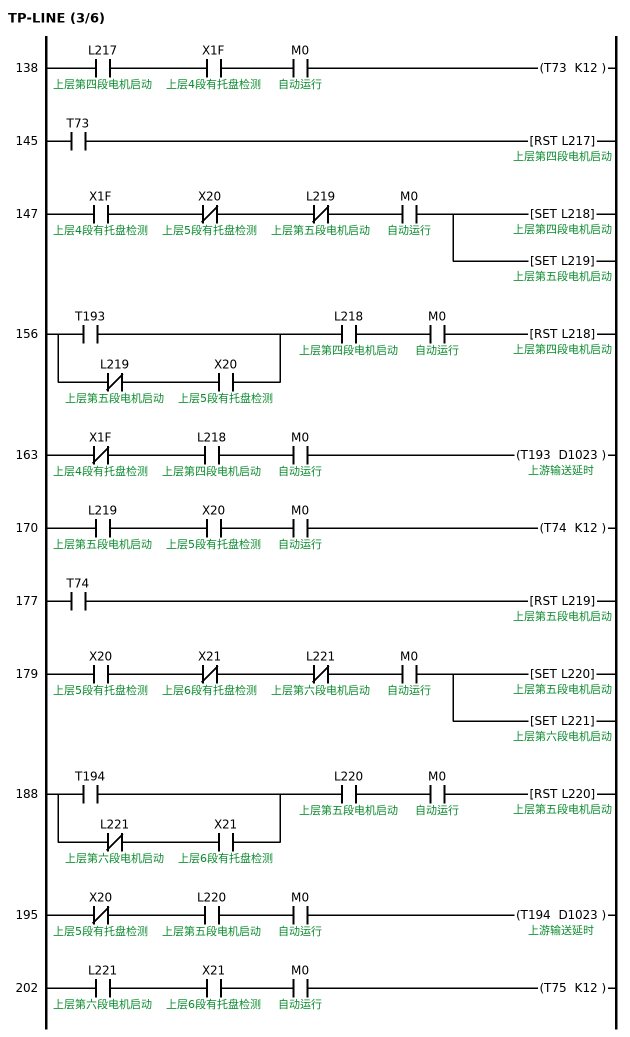
[picture p72: ladder of TP-LINE, rungs at steps 138 to 202]
138   LD      L217  ; 上层第四段电机启动
      AND     X1F  ; 上层4段有托盘检测
      AND     M0  ; 自动运行
      OUT     T73 K12
145   LD      T73
      RST     L217  ; 上层第四段电机启动
147   LD      X1F  ; 上层4段有托盘检测
      ANI     X20  ; 上层5段有托盘检测
      ANI     L219  ; 上层第五段电机启动
      AND     M0  ; 自动运行
      SET     L218  ; 上层第四段电机启动
        [note] 5
      SET     L219  ; 上层第五段电机启动
156   LD      T193
      LDI     L219  ; 上层第五段电机启动
      AND     X20  ; 上层5段有托盘检测
      ORB
      AND     L218  ; 上层第四段电机启动
      AND     M0  ; 自动运行
      RST     L218  ; 上层第四段电机启动
163   LDI     X1F  ; 上层4段有托盘检测
      AND     L218  ; 上层第四段电机启动
      AND     M0  ; 自动运行
      OUT     T193 D1023  ; 上游输送延时
170   LD      L219  ; 上层第五段电机启动
      AND     X20  ; 上层5段有托盘检测
      AND     M0  ; 自动运行
      OUT     T74 K12
177   LD      T74
      RST     L219  ; 上层第五段电机启动
179   LD      X20  ; 上层5段有托盘检测
      ANI     X21  ; 上层6段有托盘检测
      ANI     L221  ; 上层第六段电机启动
      AND     M0  ; 自动运行
      SET     L220  ; 上层第五段电机启动
        [note] 6
      SET     L221  ; 上层第六段电机启动
188   LD      T194
      LDI     L221  ; 上层第六段电机启动
      AND     X21  ; 上层6段有托盘检测
      ORB
      AND     L220  ; 上层第五段电机启动
      AND     M0  ; 自动运行
      RST     L220  ; 上层第五段电机启动
195   LDI     X20  ; 上层5段有托盘检测
      AND     L220  ; 上层第五段电机启动
      AND     M0  ; 自动运行
      OUT     T194 D1023  ; 上游输送延时
202   LD      L221  ; 上层第六段电机启动
      AND     X21  ; 上层6段有托盘检测
      AND     M0  ; 自动运行
      OUT     T75 K12
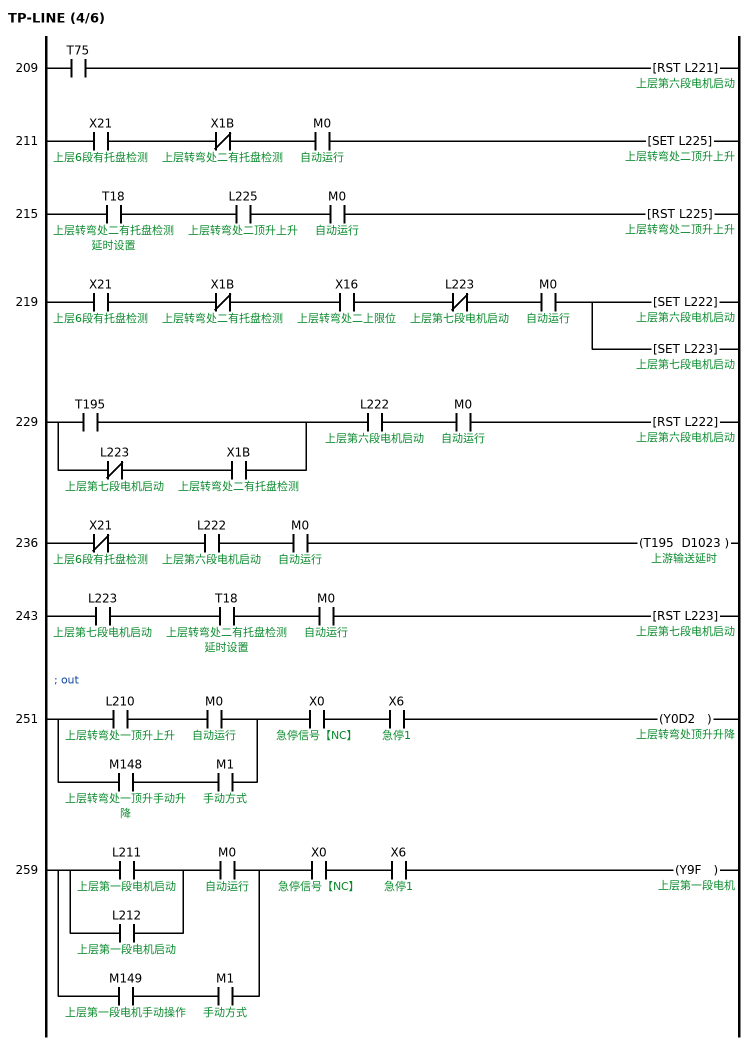
209   LD      T75
      RST     L221  ; 上层第六段电机启动
211   LD      X21  ; 上层6段有托盘检测
      ANI     X1B  ; 上层转弯处二有托盘检测
      AND     M0  ; 自动运行
      SET     L225  ; 上层转弯处二顶升上升
215   LD      T18  ; 上层转弯处二有托盘检测延时设置
      AND     L225  ; 上层转弯处二顶升上升
      AND     M0  ; 自动运行
      RST     L225  ; 上层转弯处二顶升上升
219   LD      X21  ; 上层6段有托盘检测
      ANI     X1B  ; 上层转弯处二有托盘检测
      AND     X16  ; 上层转弯处二上限位
      ANI     L223  ; 上层第七段电机启动
      AND     M0  ; 自动运行
      SET     L222  ; 上层第六段电机启动
        [note] 7
      SET     L223  ; 上层第七段电机启动
229   LD      T195
      LDI     L223  ; 上层第七段电机启动
      AND     X1B  ; 上层转弯处二有托盘检测
      ORB
      AND     L222  ; 上层第六段电机启动
      AND     M0  ; 自动运行
      RST     L222  ; 上层第六段电机启动
236   LDI     X21  ; 上层6段有托盘检测
      AND     L222  ; 上层第六段电机启动
      AND     M0  ; 自动运行
      OUT     T195 D1023  ; 上游输送延时
243   LD      L223  ; 上层第七段电机启动
      AND     T18  ; 上层转弯处二有托盘检测延时设置
      AND     M0  ; 自动运行
      RST     L223  ; 上层第七段电机启动
; out
251   LD      L210  ; 上层转弯处一顶升上升
      AND     M0  ; 自动运行
      LD      M148  ; 上层转弯处一顶升手动升降
      AND     M1  ; 手动方式
      ORB
      AND     X0  ; 急停信号【NC】
      AND     X6  ; 急停1
      OUT     Y0D2  ; 上层转弯处顶升升降
259   LD      L211  ; 上层第一段电机启动
      OR      L212  ; 上层第一段电机启动
      AND     M0  ; 自动运行
      LD      M149  ; 上层第一段电机手动操作
      AND     M1  ; 手动方式
      ORB
      AND     X0  ; 急停信号【NC】
      AND     X6  ; 急停1
      OUT     Y9F  ; 上层第一段电机
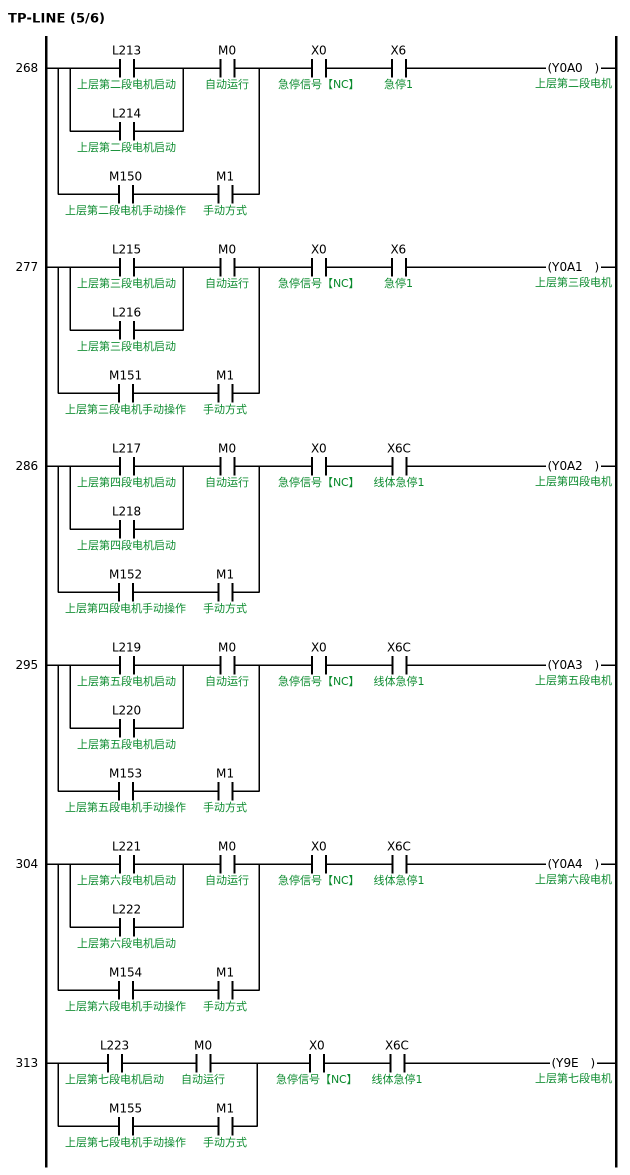
268   LD      L213  ; 上层第二段电机启动
      OR      L214  ; 上层第二段电机启动
      AND     M0  ; 自动运行
      LD      M150  ; 上层第二段电机手动操作
      AND     M1  ; 手动方式
      ORB
      AND     X0  ; 急停信号【NC】
      AND     X6  ; 急停1
      OUT     Y0A0  ; 上层第二段电机
277   LD      L215  ; 上层第三段电机启动
      OR      L216  ; 上层第三段电机启动
      AND     M0  ; 自动运行
      LD      M151  ; 上层第三段电机手动操作
      AND     M1  ; 手动方式
      ORB
      AND     X0  ; 急停信号【NC】
      AND     X6  ; 急停1
      OUT     Y0A1  ; 上层第三段电机
286   LD      L217  ; 上层第四段电机启动
      OR      L218  ; 上层第四段电机启动
      AND     M0  ; 自动运行
      LD      M152  ; 上层第四段电机手动操作
      AND     M1  ; 手动方式
      ORB
      AND     X0  ; 急停信号【NC】
      AND     X6C  ; 线体急停1
      OUT     Y0A2  ; 上层第四段电机
295   LD      L219  ; 上层第五段电机启动
      OR      L220  ; 上层第五段电机启动
      AND     M0  ; 自动运行
      LD      M153  ; 上层第五段电机手动操作
      AND     M1  ; 手动方式
      ORB
      AND     X0  ; 急停信号【NC】
      AND     X6C  ; 线体急停1
      OUT     Y0A3  ; 上层第五段电机
304   LD      L221  ; 上层第六段电机启动
      OR      L222  ; 上层第六段电机启动
      AND     M0  ; 自动运行
      LD      M154  ; 上层第六段电机手动操作
      AND     M1  ; 手动方式
      ORB
      AND     X0  ; 急停信号【NC】
      AND     X6C  ; 线体急停1
      OUT     Y0A4  ; 上层第六段电机
313   LD      L223  ; 上层第七段电机启动
      AND     M0  ; 自动运行
      LD      M155  ; 上层第七段电机手动操作
      AND     M1  ; 手动方式
      ORB
      AND     X0  ; 急停信号【NC】
      AND     X6C  ; 线体急停1
      OUT     Y9E  ; 上层第七段电机
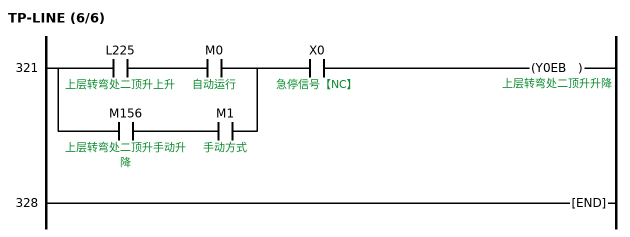
321   LD      L225  ; 上层转弯处二顶升上升
      AND     M0  ; 自动运行
      LD      M156  ; 上层转弯处二顶升手动升降
      AND     M1  ; 手动方式
      ORB
      AND     X0  ; 急停信号【NC】
      OUT     Y0EB  ; 上层转弯处二顶升升降
328   END
END_PROGRAM

PROGRAM ServoScan
VAR
  istep : INT;  (* 扫码步骤 *)
END_VAR
VAR CONSTANT
  ROW : INT := 8;  (* Y轴每个值对应的电池数量 *)
END_VAR
VAR
  ii : INT;
  jj : INT;
  m_xclean : BOOL;  (* 清零 *)
  kk : INT;  (* 错误位 *)
END_VAR

(*报警信息读取*)
g_iXanisAlarm:=U10\G806;
g_iYanisAlarm:=U10\G906;
(*报警复位*)
IF LDP(TRUE,g_xResetServo) THEN
	U10\G1502:=1;(*X轴复位*)(*这俩信号都能自动复位*)
	U10\G1602:=1;(*Y轴复位*)
	U10\G1503:=1;(*X轴重起*)
	U10\G1603:=1;(*Y轴重起*)
	YBE:= X78 OR  X79;(*X78,X79为两个驱动器的报警，这个驱动器只能断电复位，所以YAE控制断电*)
ELSIF LDF(TRUE,g_xResetServo)THEN
	YBE:=0;
END_IF;	







(*下面是正式流程*)
(*除了正常运过去那种，有时手动放上去的也要能启动扫码流程，要加个按钮*)
SET( g_xPutInto, g_xServoStart );
 CASE istep OF 
 0:(*初始化，等待启动信号*)
 				IF NOT g_xQD75Busy1 AND NOT g_xQD75Busy2 THEN
 							U10\G1500:=9001;(*9001表示会回原点*)
 							U10\G1600:=9001;
 							g_yQD75LocateStart1:=NOT g_xQD75Error1 AND NOT g_xResetServo;
 							g_yQD75LocateStart2:=NOT g_xQD75Error2 AND NOT g_xResetServo;
 				END_IF;			
 				MOV( g_xServoStart AND U10\G800=0 AND U10\G900=0, 10, istep );(*800是当前位置值*)
 	(*10是在0之后，1之前的一个步骤，扫框码，等待扫码完成。懒得改，就插在这里了*)
 10:(*扫框码，扫码完成再去扫电池码*)
 				(*夹紧气缸夹住*)
 				g_yQD75LocateStart1:=0;
 				g_yQD75LocateStart2:=0;
 				g_xCatchCylinder:=1;
 	 			g_xServoStart:=0;
 				g_xScan:=0; 	
 				D3000:=2;(**扫框码请求**)
 				IF D2000=2 THEN(*扫码成功*)
 							g_iXaxisNumber:=1;
 							g_iYaxisNumber:=1;
 							istep:=1;
 				END_IF;	
 1:(*伺服行走*)
 				(*X轴行走*)	
 				IF NOT g_xQD75LocateDone1 AND g_iXaxisNumber<>0 THEN(*起始地址设定是100，那么g_xQD75LocateDone1就是1轴定位完成信号*)
 							U10\G1500:=g_iXaxisNumber;(*起始地址设定是100，这里就要写U10，起始地址去掉个0。G1500是X轴定位启动的编号*)
 							g_yQD75LocateStart1:=NOT g_xQD75Error1;(*起始地址设定是100，那么g_yQD75LocateStart1就是1轴定位启动信号*)
 				ELSE
 							U10\G1500:=0;
 							g_yQD75LocateStart1:=0;
 				END_IF;		
 				(*Y轴行走*)	
 				IF NOT g_xQD75LocateDone2 AND g_iYaxisNumber<>0 THEN
 							U10\G1600:=g_iYaxisNumber;
 							g_yQD75LocateStart2:=NOT g_xQD75Error2;
 				ELSE
 							U10\G1600:=0;
 							g_yQD75LocateStart2:=0;
 				END_IF;	
 				SET( g_xQD75LocateDone1 AND g_xQD75LocateDone2 , g_xScan);
 				MOV( g_xQD75LocateDone1 AND g_xQD75LocateDone2 , 2, istep );
 2:(*进行扫码*)
 				g_yQD75LocateStart1:=0;
 				g_yQD75LocateStart2:=0;
 				(*扫码结果为8，表示扫码错误，调回step1，重新扫一次*)
 				IF g_iBatteryInformation[0]=8 AND TS67 THEN
 							g_iBatteryInformation[0]:=0;
 							g_xScan:=0;
 							IF  g_iXaxisNumber<20 THEN(*表示第一次扫码尝试失败*)
 										g_iXaxisNumber:=g_iXaxisNumber+20;
 										g_iYaxisNumber:=g_iYaxisNumber+20;
 										istep:=1;
 							ELSIF g_iXaxisNumber>20 THEN(*表示第二次扫码失败，两次都扫失败就跳过了*)
 										FOR ii:=0 TO 10 DO
 													IF g_iScanError[ii]=0 THEN(*把错误字都存起来，完成任务清零*)
 															g_iScanError[ii]:=g_iBatteryPosition;
 															EXIT;
 													END_IF;
 										END_FOR;	
 										IF g_iBatteryPosition>0 AND g_iBatteryPosition<128 THEN	
 													g_iBatteryPosition:=g_iBatteryPosition+1;
 													g_iYaxisNumber:=(g_iBatteryPosition-1)/ROW+1;
 													g_iXaxisNumber:=2*((g_iBatteryPosition-1)MOD ROW)+1+((g_iYaxisNumber-1) MOD 2);(*后面这个是判断奇偶的，奇数列不加，偶数列加1*)
 													istep:=1;
 										ELSIF g_iBatteryPosition=128	THEN
 													istep:=3;
 										END_IF;			
 							END_IF;	
 				END_IF;	
 				Z0:=(g_iBatteryPosition-1)*15;(*正常情况，每个电池占用15个字,-1是因为位置参数是从1开始，不是0开始*)
 				IF g_xScan AND g_iBatteryInformation[0]=24 THEN(*扫码成功会有24个字，不成功会有8个字，还可能读错，就会超过24个字，都属于不正常*)
 							D3006Z0:=g_iBatteryInformation[1];
 							D3007Z0:=g_iBatteryInformation[2];(*1-14都是电池码*)
 							D3008Z0:=g_iBatteryInformation[3];
 							D3009Z0:=g_iBatteryInformation[4];
 							D3010Z0:=g_iBatteryInformation[5];
 							D3011Z0:=g_iBatteryInformation[6];
 							D3012Z0:=g_iBatteryInformation[7];
 							D3013Z0:=g_iBatteryInformation[8];
 							D3014Z0:=g_iBatteryInformation[9];
 							D3015Z0:=g_iBatteryInformation[10];
 							D3016Z0:=g_iBatteryInformation[11];
 							D3017Z0:=g_iBatteryInformation[12];
 							D3018Z0:=g_iBatteryInformation[13];
 							D3019Z0:=g_iBatteryInformation[14];
 							D3020Z0:=g_iBatteryInformation[15];
 							IF g_iBatteryPosition>0 AND g_iBatteryPosition<128 AND TS67 THEN
 										g_xScan:=0;
 										(*数据复位*)
 										FOR jj:=0 TO 15 DO
 													g_iBatteryInformation[jj]:=0;
 										END_FOR;
 										(*这里的框是特殊形状的，有16列，每列对应8排，但是基数列和偶数列又是错开的，所以单独写的位置计算*)
 				 						g_iBatteryPosition:=g_iBatteryPosition+1;
 										g_iYaxisNumber:=(g_iBatteryPosition-1)/ROW+1;
 										g_iXaxisNumber:=2*((g_iBatteryPosition-1)MOD ROW)+1+((g_iYaxisNumber-1) MOD 2);(*后面这个是判断奇偶的，奇数列不加，偶数列加1*)
 										istep:=1;
 							ELSIF g_iBatteryPosition=128 AND TS67 THEN
 										g_xScan:=0;
 										istep:=3;	
 							END_IF;(*位置在1-128之间那个if*)
 				END_IF;(*扫码成功那个if*)		
 3:(*数据上传*)
 				D3001:=2;(*装载完成，数据上传*)
 				IF D2001=2 THEN(*表示数据收到，可以放行*)
 							istep:=4;
 				END_IF;
 4:(*数据复位，下料，回0步*)
 				D3001:=1;
 				g_xCatchCylinder:=0;
 				g_xScanDone:=1;
 				IF X100 THEN
 							U10\G1500:=1;
 							U10\G1600:=1;
 							g_yQD75LocateStart1:=NOT g_xQD75LocateDone1 AND NOT g_xQD75Error1;
 							g_yQD75LocateStart2:=NOT g_xQD75LocateDone2 AND NOT g_xQD75Error2;
 				END_IF;
 20:(*这里加一个专门去不良位的，调试用*)
 				 D2009:=g_iScanError[0]+g_iScanError[1](*这个没有意义，只是为了方便我看没扫上的那些位置*)
 								+g_iScanError[2]+g_iScanError[3]+g_iScanError[ 4]
								+g_iScanError[5] +g_iScanError[6] +g_iScanError[7]
  								+g_iScanError[8]+g_iScanError[9];
 				g_iYaxisNumber:=(kk-1)/ROW+1;
 				g_iXaxisNumber:=2*((kk-1)MOD ROW)+1+((g_iYaxisNumber-1) MOD 2);
 				U10\G1500:=g_iXaxisNumber;
 				U10\G1600:=g_iYaxisNumber; 
 				DMOV(TRUE,100,U10\G1518);
 				DMOV(TRUE,100,U10\G1618);
 				g_yQD75LocateStart1:=NOT g_xQD75LocateDone1 AND NOT g_yQD75JogCW1 AND NOT g_yQD75JogCCW1;
 				g_yQD75LocateStart2:=NOT g_xQD75LocateDone2 AND NOT g_yQD75JogCW2 AND NOT g_yQD75JogCCW2;
 				g_yQD75JogCW1:=NOT g_yQD75JogCCW1 AND g_xJogXCW;(*1轴JOG正转*)
 				g_yQD75JogCCW1:=NOT g_yQD75JogCW1 AND g_xJogXCCW;(*1轴JOG反转*)
 				g_yQD75JogCW2:=NOT g_yQD75JogCCW2 AND g_xJogYCW;(*2轴JOG正转*)
 				g_yQD75JogCCW2:=NOT g_yQD75JogCW2 AND g_xJogYCCW;(*2轴JOG反转*)
 				
 END_CASE;
(*这个写在case外边，方便复位*) 
IF TS190 AND NOT g_xQD75Busy1 AND NOT g_xQD75Busy2 THEN
	(*T190是下料时，离开开关延时，离开开关这么久就认为物料已远走，可以开始运下一个了*)
										(*10C和10D分别是两轴BUSY信号*)
 			FOR Z1:=0 TO 1920 DO(*物料送走，数据复位*)
 						D3006Z1:=0;
 		 	END_FOR;
 		  	D3000:=1;(*扫框码请求复位*)
 			g_xScanDone:=0;
 			g_iBatteryPosition:=1;
 			istep:=0;
END_IF;
 OUT_T( g_iBatteryInformation[0]<>0 AND istep=2,TC67 ,k1);(*扫码成功到接收数据完毕需要时间，所以做个延时*)
 OUT_T( g_iBatteryInformation[0]=0 AND istep=2 ,TC66 ,k100);(*有时候扫码请求发出去数据没接收到，需要重新启动扫码，等10S*)
 IF TS190 OR m_xclean THEN
 	FOR jj:=0 TO 9 DO
 		g_iScanError[jj]:=0;
 	END_FOR;
 END_IF;
END_PROGRAM

PROGRAM TCP
VAR
  m_tonReconnect : TON;  (* 自动重连 *)
  m_xReconnect : BOOL;
  m_tReconnectCurrentTime : TIME;
  m_tonAutoClose : TON;  (* 自动关闭 *)
  m_xAutoClose : BOOL;
  m_tAutoCloseCurrentTime : TIME;
  m_ton1ReceiveHeartbeat : TON;  (* 心跳检查 *)
  m_t1RecHeartbeatCurrentTime : TIME;
  m_xOpenSuccess : BOOL;  (* 打开成功 *)
  m_xSendSuccess : BOOL;  (* 发送成功 *)
  m_xReceiveSuccess : BOOL;  (* 接收成功 *)
  m_iOpenCtrl : INT;  (* 打开指令控制字 *)
  m_iSendCtrl : INT;  (* 发送指令控制字 *)
  m_iReceivectrl : INT;  (* 接收指令控制字 *)
  m_iClosectrl : INT;  (* 关闭指令控制字 *)
  m_xCloseSuccess : BOOL;  (* 关闭成功 *)
END_VAR
D200:=4;
D201:=H54;(*16进制的54就是T，扫码枪设定的扫码触发条件*)
m_tonReconnect(IN:= NOT SD1282.0 AND NOT SD1284.0  ,PT:=T#5s  ,Q:=m_xReconnect ,ET:=m_tReconnectCurrentTime);
SP_SOCOPEN(m_xReconnect  AND SD1288.A , "U0", K1 , D100, M900);
SP_SOCSND( LDP(TRUE,g_xScan) AND SD1282.0 , "U0" , K1 , D110, D200, M910);
SP_SOCRCV( SD1282.0 AND SD1286.0 AND NOT M920, "U0" , K1, D120, g_iBatteryInformation[0],M920);
m_tonAutoClose(IN:= SD1284.0 AND NOT SD1282.0 ,PT:=T#5s,Q:=m_xAutoClose ,ET:= m_tAutoCloseCurrentTime );
SP_SOCCLOSE( LDF(TRUE,SD1282.0) OR m_xAutoClose  , "U0" , K1, D130, M930);
END_PROGRAM

// device comments not shown above
X7  ; 急停2
X6D  ; 线体急停2
X0B2  ; 上层开门信号
X0B3  ; 下层开门信号
X0B4  ; 下层出货完成信号
Y0B8  ; 扫码位置阻挡
M52  ; 无原点提示
L60  ; 工位1-2送出输送速度
L140  ; 工位3-2送出输送速度
L224  ; 上层第七段电机启动
L226  ; 上层第三段电机启动
L227  ; 上层第二段电机启动
L252  ; 下层第十一段电机启动
T0  ; AB门上层出口段托盘到位无货延时
D436  ; 出口待机时间
D438  ; 上料待机时间
D456  ; 运行时间（分）
D522  ; 出口待机时间（分）
D534  ; 工作时间
D536  ; 故障率
D540  ; 稼动率
D544  ; 节拍
D550  ; 故障时间
D554  ; 运行-待机
D560  ; 工作时间
D564  ; 运行时间
D800  ; 延时时间设置
D801  ; 减速时间设定
D1051  ; AB门输送报警延时设置
